PROGRAM PackMLExample
VAR
	example: ExampleStateMachine;
	
	iStateResult: I_State;
	iSmgr: I_StateManager;
	bError: BOOL;
	bInit: BOOL := TRUE;
	
	
	sStateToRequest: Str := '*.idle'; // Use this variable to tell program which state to request
	bRequest: BOOL; // Rising edge will trigger the state change.
	
END_VAR

IF bInit THEN
	bInit := FALSE;
	bError := IsFail(GetStateManager(example.Entity, iSmgr));
END_IF

IF bError THEN
	RETURN;
END_IF

IF NOT bRequest THEN
	RETURN;
END_IF

bRequest := FALSE;

IF IsOk(GetState(example.Entity, sStateToRequest, iStateResult)) THEN
	iSmgr.Request(iStateResult);
END_IF

END_PROGRAM

(* stored: Version 1.1.0.1
   POU PackMLExample: Id {666c2c12-90f3-4c2d-9ee4-20e6b6ddb464}, SpecialFunc None *)
